Staubli VAL3: message.pgx

public program message(string& message[], num index)
// English IF message
begin
  // lenght of message
  //
  switch index
    case 0
      message="你要进入:"
    break
    case 1
      message="< IF 向导 >"
    break
    case 2
      message="选择条件类型"
    break
    case 3
      message="选择输入"
    break
    case 4
      message="选择输出"
    break
    case 5
      message="选择EMAP输入"
    break
    case 6
      message="选择运行指令的方式"
    break
    case 7
      message="选择指令来关联:"
    break
    case 8
      message="从列表中选择: "
    break
  endSwitch
end
